FUNCTION_BLOCK FB_OperatingMode
//---------------------------------------------------------------------------------------------------------------
//
//  Fen 2023.12.21
//
//  - XTS_TRAINING
//  - example project for setting up transport layer
//
//
//  FB_OperatingMode
//  - Operating Mode handler for XTS_training Exsample
//  - 
//
//
//---------------------------------------------------------------------------------------------------------------
// This SOFTWARE is provided as an Exemple by THE PROVIDER "as is" and "with all faults." THE PROVIDER makes no 
// representations or warranties of any kind concerning the safety, suitability, lack of viruses, inaccuracies, 
// typographical errors, or other harmful components of this SOFTWARE. There are inherent dangers in the use of 
// any software, and you are solely responsible for determining whether this SOFTWARE is compatible with your 
// equipment and other software installed on your equipment. You are also solely responsible for the protection 
// of your equipment and backup of your data, and THE PROVIDER will not be liable for any damages you may suffer 
// in connection with using, modifying, or distributing this SOFTWARE.
//---------------------------------------------------------------------------------------------------------------

VAR 
	_eState			: E_OperatingState;	
	_eLastState		: E_OperatingState;

	_eCommand		: E_OperatingCmd;
	_eActCommand	: E_OperatingCmd;
	

	_StaeCompleteRtrig	:R_TRIG;
	_StaeComplete		: BOOL;

	
	_bSingelStep				: BOOL;

END_VAR

PROPERTY Command : E_OperatingCmd
GET

	Command := _eActCommand;
END_GET
SET

	_eCommand := Command;
END_SET
END_PROPERTY

METHOD Cyclic
VAR_INPUT
END_VAR
// simple Example for Operatingmode handler


// State Complete
	_StaeCompleteRtrig();
	IF _StaeCompleteRtrig.Q THEN
		_StaeComplete := TRUE;
	END_IF

// Xts Operating Mode

	_eActCommand := _eActCommand;

	CASE _eState OF
	
	// Invalid 	--> wait for Cmd 	
	E_OperatingState.OperatingMode_INVALID : 
		IF _eCommand = E_OperatingCmd.OperatingCmd_Clear THEN
			_eState := E_OperatingState.OperatingMode_Clear;
			_eActCommand := E_OperatingCmd.OperatingCmd_DONE;
			_eLastState := E_OperatingState.OperatingMode_INVALID;
		
		ELSE 
			_eActCommand := E_OperatingCmd.OperatingCmd_DONE;	
		END_IF
		
	// Clear 	--> Init Ca-Group  and Axis 	
	E_OperatingState.OperatingMode_Clear:
		IF _StaeComplete 
		THEN
			_StaeComplete := FALSE;
			_eState := E_OperatingState.OperatingMode_Clear_Sc;
		END_IF
		
		CASE _eCommand	OF  			
			E_OperatingCmd.OperatingCmd_Reset :	
				_eState := E_OperatingState.OperatingMode_Reset;
				_eActCommand := E_OperatingCmd.OperatingCmd_DONE;
				_eLastState := E_OperatingState.OperatingMode_Clear;
			
		ELSE 
			_eActCommand := E_OperatingCmd.OperatingCmd_DONE;	
				
		END_CASE
		
	// Clear_Sc 	--> State complete	
	E_OperatingState.OperatingMode_Clear_Sc :
		CASE _eCommand	OF  
			E_OperatingCmd.OperatingCmd_Clear :
				_eState := E_OperatingState.OperatingMode_Clear;
				_eActCommand := E_OperatingCmd.OperatingCmd_DONE;
				_eLastState := E_OperatingState.OperatingMode_Clear_Sc;
			
			E_OperatingCmd.OperatingCmd_Reset :	
				_eState := E_OperatingState.OperatingMode_Reset;
				_eActCommand := E_OperatingCmd.OperatingCmd_DONE;
				_eLastState := E_OperatingState.OperatingMode_Clear_Sc;
				
			E_OperatingCmd.OperatingCmd_Prepare	:
				_eState := E_OperatingState.OperatingMode_Prepare;
				_eActCommand := E_OperatingCmd.OperatingCmd_DONE;
				_eLastState := E_OperatingState.OperatingMode_Clear_Sc;
		
		ELSE 
			_eActCommand := E_OperatingCmd.OperatingCmd_DONE;	
				
		END_CASE
		
	
	// Prepare 	--> build Ca-Group  and enable Axis 	
	E_OperatingState.OperatingMode_Prepare :
		IF _StaeComplete 
		THEN
			_StaeComplete := FALSE;
			_eState := E_OperatingState.OperatingMode_Prepar_Sc;
		END_IF
		
		CASE _eCommand	OF  
			E_OperatingCmd.OperatingCmd_Clear :
				_eState := E_OperatingState.OperatingMode_Clear;
				_eActCommand := E_OperatingCmd.OperatingCmd_DONE;
				_eLastState := E_OperatingState.OperatingMode_Prepare;
			
			E_OperatingCmd.OperatingCmd_Reset :	
				_eState := E_OperatingState.OperatingMode_Reset;
				_eActCommand := E_OperatingCmd.OperatingCmd_DONE;
				_eLastState := E_OperatingState.OperatingMode_Prepare;
		
		ELSE 
			_eActCommand := E_OperatingCmd.OperatingCmd_DONE;	
		END_CASE
	
	// Stopping 	--> stop Axis 		
	E_OperatingState.OperatingMode_Stopping :
		IF _StaeComplete 
		THEN
			_StaeComplete := FALSE;
			_eState := E_OperatingState.OperatingMode_Prepar_Sc;
		END_IF
		CASE _eCommand	OF  
			E_OperatingCmd.OperatingCmd_Clear :
				_eState := E_OperatingState.OperatingMode_Clear;
				_eActCommand := E_OperatingCmd.OperatingCmd_DONE;
				_eLastState := E_OperatingState.OperatingMode_Stopping;
			
			E_OperatingCmd.OperatingCmd_Reset :	
				_eState := E_OperatingState.OperatingMode_Reset;
				_eActCommand := E_OperatingCmd.OperatingCmd_DONE;
				_eLastState := E_OperatingState.OperatingMode_Stopping;
		
		ELSE 
			_eActCommand := E_OperatingCmd.OperatingCmd_DONE;	
		END_CASE
		
	// Prepare 	--> emptying the system 		
	E_OperatingState.OperatingMode_Empty:
		IF _StaeComplete 
		THEN
			_StaeComplete := FALSE;
			_eState := E_OperatingState.OperatingMode_Prepar_Sc;
		END_IF
		
		CASE _eCommand	OF  
			E_OperatingCmd.OperatingCmd_Clear :
				_eState := E_OperatingState.OperatingMode_Clear;
				_eActCommand := E_OperatingCmd.OperatingCmd_DONE;
				_eLastState := E_OperatingState.OperatingMode_Empty;
			
			E_OperatingCmd.OperatingCmd_Reset :	
				_eState := E_OperatingState.OperatingMode_Reset;
				_eActCommand := E_OperatingCmd.OperatingCmd_DONE;
				_eLastState := E_OperatingState.OperatingMode_Empty;
				
			E_OperatingCmd.OperatingCmd_Stopping :
				_eState := E_OperatingState.OperatingMode_Stopping;
				_eActCommand := E_OperatingCmd.OperatingCmd_DONE;
				_eLastState := E_OperatingState.OperatingMode_Empty;
		
		ELSE 
			_eActCommand := E_OperatingCmd.OperatingCmd_DONE;	
			
		END_CASE
	
	// 	Prepare 	--> State complete
	E_OperatingState.OperatingMode_Prepar_Sc:
		CASE _eCommand	OF  
			E_OperatingCmd.OperatingCmd_Clear :
				_eState := E_OperatingState.OperatingMode_Clear;
				_eActCommand := E_OperatingCmd.OperatingCmd_DONE;
				_eLastState := E_OperatingState.OperatingMode_Prepar_Sc;
			
			E_OperatingCmd.OperatingCmd_Reset :	
				_eState := E_OperatingState.OperatingMode_Reset;
				_eActCommand := E_OperatingCmd.OperatingCmd_DONE;
				_eLastState := E_OperatingState.OperatingMode_Prepar_Sc;
				
			E_OperatingCmd.OperatingCmd_Stopping :
				_eState := E_OperatingState.OperatingMode_Stopping;
				_eActCommand := E_OperatingCmd.OperatingCmd_DONE;
				_eLastState := E_OperatingState.OperatingMode_Prepar_Sc;
			
			E_OperatingCmd.OperatingCmd_Home 	:
				_eState := E_OperatingState.OperatingMode_Home;
				_eActCommand := E_OperatingCmd.OperatingCmd_DONE;
				_eLastState := E_OperatingState.OperatingMode_Prepar_Sc;
		
		ELSE 
			_eActCommand := E_OperatingCmd.OperatingCmd_DONE;	
	
		END_CASE
		
	// 	Empty 	--> State complete
	E_OperatingState.OperatingMode_Empty_Sc:
			_eState := E_OperatingState.OperatingMode_Prepar_Sc;
			_eLastState := E_OperatingState.OperatingMode_Empty_Sc;
		
	// 	Stopping 	--> State complete
	E_OperatingState.OperatingMode_Stopping_Sc:
			_eState := E_OperatingState.OperatingMode_Prepar_Sc;
			_eLastState := E_OperatingState.OperatingMode_Stopping_Sc;


	
	// 	Home 	--> Move to Start Position
	E_OperatingState.OperatingMode_Home :
		IF _StaeComplete 
		THEN
			_StaeComplete := FALSE;
			_eState := E_OperatingState.OperatingMode_Home_Sc;
		END_IF
		
		CASE _eCommand	OF  
			E_OperatingCmd.OperatingCmd_Clear :
				_eState := E_OperatingState.OperatingMode_Clear;
				_eActCommand := E_OperatingCmd.OperatingCmd_DONE;
				_eLastState := E_OperatingState.OperatingMode_Home;
			
			E_OperatingCmd.OperatingCmd_Reset :	
				_eState := E_OperatingState.OperatingMode_Reset;
				_eActCommand := E_OperatingCmd.OperatingCmd_DONE;
				_eLastState := E_OperatingState.OperatingMode_Home;
				
			E_OperatingCmd.OperatingCmd_Stopping :
				_eState := E_OperatingState.OperatingMode_Stopping;
				_eActCommand := E_OperatingCmd.OperatingCmd_DONE;
				_eLastState := E_OperatingState.OperatingMode_Home;
		
		ELSE 
			_eActCommand := E_OperatingCmd.OperatingCmd_DONE;	
	
		END_CASE
	
	// 	Home 	--> State complete
	E_OperatingState.OperatingMode_Home_Sc :	
		_eState := E_OperatingState.OperatingMode_Active;
		
		CASE _eCommand	OF  
			E_OperatingCmd.OperatingCmd_Clear :
				_eState := E_OperatingState.OperatingMode_Clear;
				_eActCommand := E_OperatingCmd.OperatingCmd_DONE;
				_eLastState := E_OperatingState.OperatingMode_Home_Sc;
			
			E_OperatingCmd.OperatingCmd_Reset :	
				_eState := E_OperatingState.OperatingMode_Reset;
				_eActCommand := E_OperatingCmd.OperatingCmd_DONE;
				_eLastState := E_OperatingState.OperatingMode_Home_Sc;
				
			E_OperatingCmd.OperatingCmd_Stopping :
				_eState := E_OperatingState.OperatingMode_Stopping;
				_eActCommand := E_OperatingCmd.OperatingCmd_DONE;
				_eLastState := E_OperatingState.OperatingMode_Home_Sc;
		
		ELSE 
			_eActCommand := E_OperatingCmd.OperatingCmd_DONE;	
	
		END_CASE
	
	// 	Active/Work 	--> execute work sequences
 	E_OperatingState.OperatingMode_Active :
		CASE _eCommand	OF  
			E_OperatingCmd.OperatingCmd_Clear :
				_eState := E_OperatingState.OperatingMode_Clear;
				_eActCommand := E_OperatingCmd.OperatingCmd_DONE;
				_eLastState := E_OperatingState.OperatingMode_Active;
			
			E_OperatingCmd.OperatingCmd_Reset :	
				_eState := E_OperatingState.OperatingMode_Reset;
				_eActCommand := E_OperatingCmd.OperatingCmd_DONE;
				_eLastState := E_OperatingState.OperatingMode_Active;
				
			E_OperatingCmd.OperatingCmd_Stopping :
				_eState := E_OperatingState.OperatingMode_Stopping;
				_eActCommand := E_OperatingCmd.OperatingCmd_DONE;
				_eLastState := E_OperatingState.OperatingMode_Active;
			
			E_OperatingCmd.OperatingCmd_Empty 	:
				_eState := E_OperatingState.OperatingMode_Empty;
				_eActCommand := E_OperatingCmd.OperatingCmd_DONE;
				_eLastState := E_OperatingState.OperatingMode_Active;
		
		ELSE 
			_eActCommand := E_OperatingCmd.OperatingCmd_DONE;	
				
		END_CASE
	
	// 	Reset 	--> Reset Error --> Jump to last state back
	E_OperatingState.OperatingMode_Reset :
		IF _StaeComplete 
		THEN
			_StaeComplete := FALSE;
			_eState := _eLastState;
			_eLastState := E_OperatingState.OperatingMode_Reset;
		END_IF
	
		_eActCommand := E_OperatingCmd.OperatingCmd_DONE;
		
	
	END_CASE
END_METHOD

PROPERTY eLastState : E_OperatingState
GET

	eLastState := _eLastState;
END_GET
END_PROPERTY

PROPERTY eState : E_OperatingState
GET

	eState := _eState;
END_GET
END_PROPERTY

METHOD M_StateComplete
VAR_INPUT
END_VAR

	//_StaeCompleteRtrig.CLK := TRUE;
	_StaeComplete := TRUE;
END_METHOD

PROPERTY sState : STRING
GET

	sState := to_String(_eState);
END_GET
END_PROPERTY

END_FUNCTION_BLOCK

(* stored: Version 1.1.0.1, ProductVersion 3.1.4024.12
   POU FB_OperatingMode: Id {de7b5e8c-5b1c-4a12-8318-2ed22844172c}, SpecialFunc None
   Folder methods: Id {0dc0e828-bf35-4e0b-8703-4268543de7b2}
   Folder properties: Id {8813dc4b-dc38-4062-9720-762145ef1089}
   Property Command: Id {d8f5591a-e6d3-4a29-80fb-7ae3f7322058}
   Get Get: Id {f1268c48-b36d-4a61-8162-213144ba2954}
   Set Set: Id {d428204b-ff14-4cfd-a98d-e5c5150b88f2}
   Method Cyclic: Id {d308db6f-4fba-49e2-a1b0-d7e8b95f16fb}
   Property eLastState: Id {6153c592-974e-4e4a-ae45-335c88a700cf}
   Get Get: Id {ef7f7887-7faa-4eb2-86fc-3992378158aa}
   Property eState: Id {e653646f-3c8b-4d08-8850-5be3336e0c64}
   Get Get: Id {5e0cc501-1836-47d5-a17a-cecbb9614543}
   Method M_StateComplete: Id {27eebfff-3a01-4a97-9e43-f043f4d00ba6}
   Property sState: Id {3406648a-160c-419e-b75f-bf6c7936494e}
   Get Get: Id {ff35ccfd-db26-4f17-b0ef-149128e22ad1} *)
